// TIA Portal V17 export
FUNCTION "FC_烧嘴报警" : Void   // FC, LAD
{ S7_Optimized_Access := 'TRUE' }
   VAR_TEMP   // added for the SCL form of the ladder/FBD networks
      _w1 : Bool;
      _w2 : Bool;
   END_VAR
BEGIN

REGION Network 1: 故障反馈上升沿触发蜂鸣器
   // 7路故障反馈常开触点并联，汇总后经R_TRIG上升沿检测，任意一路故障反馈从0→1时置位蜂鸣器Q4.7
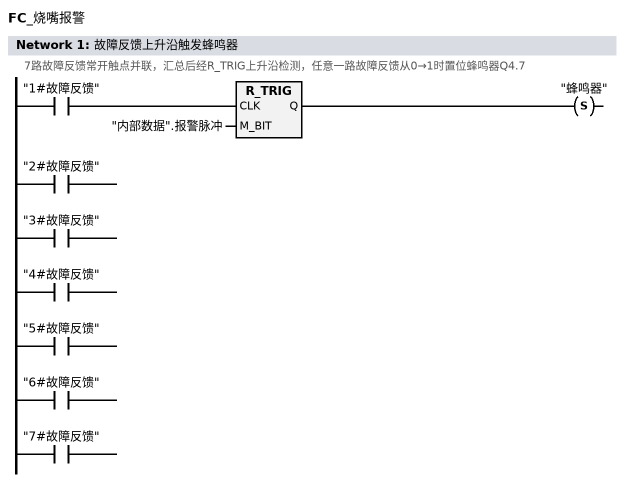
   #_w2 := "1#故障反馈";
   R_TRIG(CLK := "1#故障反馈", M_BIT := "内部数据".报警脉冲, Q => #_w1);
   IF #_w1 THEN "蜂鸣器" := TRUE; END_IF;
END_REGION
END_FUNCTION
